{attribute 'Tc2GvlVarNames'}
VAR_GLOBAL
	Axis1: Axis_Ref;
	Axis2: Axis_Ref;
	Axis3: Axis_Ref;
END_VAR

(* stored: Version 1.1.0.1, ProductVersion 3.1.4024.12
   GVL Global_Variables: Id {6920524c-a957-4a63-8efc-2c6aa8920c41} *)
